FUNCTION_BLOCK FB_DeadBand
VAR_INPUT
	fSignal : LREAL;
	fDeadBandUp : LREAL;
	fDeadBandDown : LREAL;
	fXDotRef : LREAL;
END_VAR
VAR_OUTPUT
	fCompansatedSignal : LREAL;
END_VAR
VAR
	fSignalUp : LREAL;
	fSignalDown : LREAL;
END_VAR

IF fXDotRef > 0 THEN
	fCompansatedSignal := fSignal + fDeadBandUp;
ELSIF fXDotRef < 0 THEN
	fCompansatedSignal := fSignal - fDeadBandDown;
ELSE
	fCompansatedSignal := 0.0;
END_IF

IF fCompansatedSignal < -1.0 THEN
	fCompansatedSignal := -1.0;
ELSIF fCompansatedSignal > 1.0 THEN
	fCompansatedSignal := 1.0;
ELSE
	fCompansatedSignal := fCompansatedSignal;
END_IF

END_FUNCTION_BLOCK

(* stored: Version 1.1.0.1
   POU FB_DeadBand: Id {b17f7937-cf2d-4500-9946-ab7a5f687a16}, SpecialFunc None *)
